FUNCTION_BLOCK NumberToEventAdapter_4
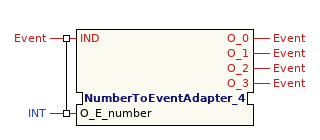
  EVENT_INPUT
    IND WITH O_E_number;
  END_EVENT
  EVENT_OUTPUT
    O_0;
    O_1;
    O_2;
    O_3;
  END_EVENT
  VAR_INPUT
    O_E_number : INT;
  END_VAR
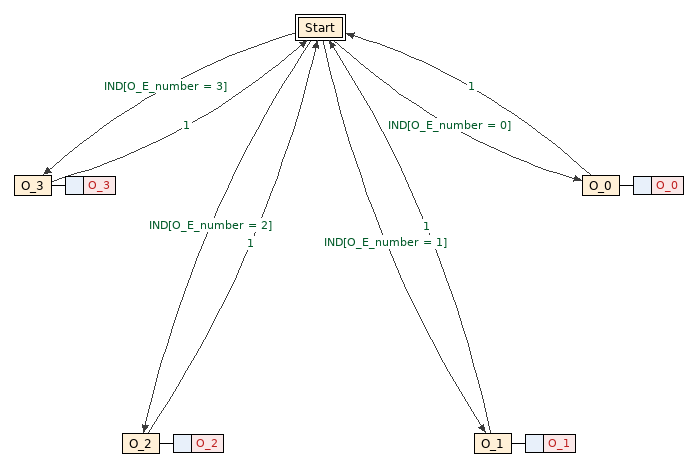
  EC_STATES
    Start;
    O_0 : -> O_0;
    O_1 : -> O_1;
    O_2 : -> O_2;
    O_3 : -> O_3;
  END_STATES
  EC_TRANSITIONS
    Start TO O_0 := IND[O_E_number = 0];
    O_0 TO Start := 1;
    Start TO O_1 := IND[O_E_number = 1];
    O_1 TO Start := 1;
    Start TO O_2 := IND[O_E_number = 2];
    O_2 TO Start := 1;
    Start TO O_3 := IND[O_E_number = 3];
    O_3 TO Start := 1;
  END_TRANSITIONS
END_FUNCTION_BLOCK
